{attribute 'qualified_only'}
VAR_GLOBAL
	
	//Laitteistoon liitetyt globaalit muuttujat:
	//Tulot:
	safetyOk			: BOOL := TRUE;
	start 	AT%I*		: BOOL;
	stop	AT%I*	 	: BOOL;
	playCW	AT%I*		: BOOL;
	playCCW	AT%I*		: BOOL;
	tila1	AT%I*		: BOOL;
	tila2	AT%I*		: BOOL;
	reset	AT%I*		: BOOL;
	//stepperSpeed	: INT := 0;
	
	//GUI
	
	startGUI 			: BOOL;
	stopGUI				: BOOL;
	resetGUI			: BOOL;
	asemannollausGUI 	: BOOL;
	triggerGUI			: BOOL;

	//Lähdöt:

	systemOnLight		AT%Q*	: BOOL;
	safetyOkLight		AT%Q*	: BOOL;
	startBtnLight		AT%Q*	: BOOL;
	stopBtnLight		AT%Q*	: BOOL;
	resetBtnLight		AT%Q*	: BOOL;
	playCWBtnLight		AT%Q*	: BOOL;
	playCCWBtnLight		AT%Q*	: BOOL;
	
	//Muut globaalit muuttujat:
	
	driverMode		: INT := 0;
	vikamuisti		: BOOL := TRUE;
	blinker1000ms	: BOOL;
	muuVika			: BOOL;	
	systemOn		: BOOL;
	
END_VAR

(* stored: Version 1.1.0.1, ProductVersion 3.1.4024.11
   GVL GVL: Id {4975a585-f788-453e-9391-6aa63f206255} *)
